FUNCTION_BLOCK FB_UnistatControl
VAR_INPUT
	UnistatRef 		: REFERENCE TO FB_HwRefUnistat;
	nTempSetpoint 	: DINT;
	bTempControlOn	: BOOL;
	bExecute		: BOOL;
END_VAR
VAR_OUTPUT
	bBusy			: BOOL;
	bError			: BOOL;
	nErrorID		: ERRORID;
END_VAR
VAR
	fbSendCmd 		: FB_Unistat_SendCmd;
	nState			: UINT;
END_VAR

IF bExecute THEN
	IF NOT __ISVALIDREF(UnistatRef) THEN
		{warnig 'Implement proper ErrorID'}
		bError := TRUE;
		nErrorID := 333;
		RETURN;
	END_IF
	fbSendCmd.SerialPort REF= UnistatRef.P_SerialPort;
 	UnistatRef.P_bPolling := FALSE;
	
	IF nState = 0 THEN
		IF UnistatRef.P_eState = E_UnistatState.Error THEN
			RETURN;
		END_IF
		IF bTempControlOn THEN
			IF UnistatRef.P_eState = E_UnistatState.On THEN
				nState := 3;
			ELSE
				nState := 1;
			END_IF
		ELSE
			IF UnistatRef.P_eState = E_UnistatState.On THEN
				nState := 2;
			ELSE
				RETURN;
			END_IF
		END_IF
		bBusy := TRUE;
	END_IF
	
	CASE nState OF
		1:	//Ein
			fbSendCmd(bExecute:= TRUE, eCommand:= E_Unitstat_Command.Start_TempControl);
			IF NOT fbSendCmd.bBusy THEN
				fbSendCmd(bExecute:= FALSE);
				nState := 3;
			END_IF
		
		2:	//Aus
			fbSendCmd(bExecute:= TRUE, eCommand:= E_Unitstat_Command.Stop_TempControl);
			IF NOT fbSendCmd.bBusy THEN
				fbSendCmd(bExecute:= FALSE);
				bBusy := FALSE;
				nState := 80;
			END_IF
		
		3:	//Solltemperatur
			fbSendCmd(bExecute:= TRUE, eCommand:= E_Unitstat_Command.Set_TempSetPoint, nSendData := nTempSetPoint);
			IF NOT fbSendCmd.bBusy THEN
				fbSendCmd(bExecute:= FALSE);
				bBusy := FALSE;
				nState := 80;
			END_IF
	END_CASE
ELSE
	IF __ISVALIDREF(UnistatRef) THEN
		UnistatRef.P_bPolling := TRUE;
	END_IF
	nState := 0;
	bBusy := FALSE;
	bError := FALSE;
	nErrorID := 0;
END_IF

END_FUNCTION_BLOCK

(* stored: Version 1.1.0.1, ProductVersion 3.1.4024.6
   POU FB_UnistatControl: Id {661dadb5-7df8-45b5-a1c8-b3e4d15b0b85}, SpecialFunc None *)
